// Mitsubishi GX Works2 project: ethernet_config   PLC: Q02/Q02H

PROGRAM MAIN
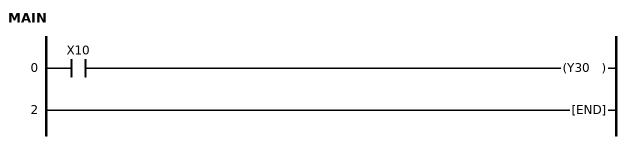
0     LD      X10
      OUT     Y30
2     END
END_PROGRAM
